PROGRAM ExtractiveOutletValveParameterMenuBindings
VAR PERSISTENT
	extractionValveParameters : ST_ExtractiveControlValveParameters;
	calibrationTimeTextField_TextVariable : DINT;
	fullOpenTimeTextField_TextVariable : DINT;
END_VAR
VAR
END_VAR


extractionValveParameters.calibrationTimeMs := calibrationTimeTextField_TextVariable;
extractionValveParameters.timeToFullyOpenMs := fullOpenTimeTextField_TextVariable;

ReactorLevelAndPressure.ExtractiveControlValveParameters := extractionValveParameters;

END_PROGRAM

(* stored: Version 1.1.0.1, ProductVersion 3.1.4024.9
   POU ExtractiveOutletValveParameterMenuBindings: Id {e0e1f055-7792-4626-bb90-c0508d8abc71}, SpecialFunc None *)
